PROGRAM INDEXING
VAR
	bStartInput : BOOL;
	bServoOn : BOOL;
	bProgram0_On : BOOL;
	bProgram1_On : BOOL :=TRUE;
	bProgram2_On : BOOL :=FALSE;
	bProgram3_On : BOOL:=FALSE;
	bProgram4_On : BOOL:=FALSE;	
	bHomePositionReturn : BOOL;
	bResetInput : BOOL;
	bEmergencyInput : BOOL := TRUE;
	
	IN_POSITION_INPUT: BOOL;
	IN_POSITIONING_COMPLETION: BOOL;
	IN_START_INPUT_WAIT: BOOL;
	IN_ALARM1: BOOL;
	IN_ALARM2: BOOL;
	IN_READY_STATE: BOOL;
	T1: TON;
	TMR1: TON;
	TMR2: TON;
	TMR3: TON;
	TMR4: TON;
	TMR5: TON;
	TMR6: TON;
	TMR7: TON;
	IN_SERVO_STATUS: BOOL;
	bFirstDigit: BOOL;
	CNT1: CTU;
	ResetCount: BOOL;
	IPC: TP;
	IN_POSITIONING_COMPLET: BOOL;
	CNT2: CTU;
	START_STRAIGTHEN: BOOL;

	START_STRAIGHTEN: R_TRIG;
	START_ROTATING: R_TRIG;
	START_ROTATION: TP;
	SS: R_TRIG;
	CNT_START: CTU;
	TMR_PROCESS: TOF;
	TMR8: TON;
	TMR_OFF: TON;
	TMR_RELEASE: TON;
	INPOS: R_TRIG;
	A: BOOL;
END_VAR

INDEXING_1_VAR.DataByteOutput[0].0 := bProgram0_On;
INDEXING_1_VAR.DataByteOutput[0].1 := bProgram1_On;
INDEXING_1_VAR.DataByteOutput[0].2 := bProgram2_On;
INDEXING_1_VAR.DataByteOutput[0].3 := bProgram3_On;
INDEXING_1_VAR.DataByteOutput[0].4 := bProgram4_On;
INDEXING_1_VAR.DataByteOutput[0].6 := bResetInput;
INDEXING_1_VAR.DataByteOutput[0].7 := bHomePositionReturn;
INDEXING_1_VAR.DataByteOutput[1].0 := bStartInput;
INDEXING_1_VAR.DataByteOutput[1].1 := bServoOn;
INDEXING_1_VAR.DataByteOutput[1].2 := bFirstDigit;
INDEXING_1_VAR.DataByteOutput[1].4 := bEmergencyInput;

IN_POSITION_INPUT := 			INDEXING_1_VAR.DataByteInput [1].0;
IN_POSITIONING_COMPLETION := 	INDEXING_1_VAR.DataByteInput [1].1;
IN_START_INPUT_WAIT := 			INDEXING_1_VAR.DataByteInput [1].2;
IN_ALARM1 := 					INDEXING_1_VAR.DataByteInput [1].3;
IN_ALARM2 := 					INDEXING_1_VAR.DataByteInput [1].4;
IN_READY_STATE :=				INDEXING_1_VAR.DataByteInput [1].7;
IN_SERVO_STATUS :=				INDEXING_1_VAR.DataByteInput [1].6; 
(*
//SERVO ON
IF NOT IN_SERVO_STATUS THEN
	bResetInput := TRUE;
	TMR4(IN:=bResetInput,PT:=T#0.5S);
	IF TMR4.Q THEN
		bResetInput := FALSE;
	END_IF
	bServoOn:=TRUE;
	//POWER_CONTROL.O_PWR_CTRL_INDEXING_1:=TRUE;
	TMR8(IN:=POWER_CONTROL.O_PWR_CTRL_INDEXING_1,PT:=T#0.5S);	
	IF TMR8.Q THEN
		POWER_CONTROL.O_PWR_CTRL_INDEXING_1:=FALSE;
		TMR8(IN:=FALSE);
	END_IF
END_IF
*)
//ALARM RESET
IF NOT IN_ALARM1 OR NOT IN_ALARM2 THEN
	bResetInput := TRUE;
	TMR4(IN:=bResetInput,PT:=T#0.5S);
	INPUT_VAR.ALARM1:=NOT IN_ALARM1 OR NOT IN_ALARM2;
	IF TMR4.Q THEN
		bResetInput := FALSE;
	END_IF
ELSE
	TMR4(IN:=FALSE);
END_IF

IF INDEXING_1_VAR.I_INDEXING_1_ROTATION_DONE THEN
		INDEXING_1_VAR.I_INDEXING_1_HOME:=TRUE;
		bHomePositionReturn:=FALSE;
		//INDEXING_1_VAR.I_INDEXING_1_ROTATION_DONE:=TRUE;
END_IF
//homing
IF NOT INDEXING_1_VAR.I_INDEXING_1_HOME THEN
	bHomePositionReturn:=TRUE;
 	ResetCount:=TRUE;
	INDEXING_1_VAR.O_ROTATION_START:=FALSE;
	INDEXING_1_VAR.I_INDEXING_1_ROTATION_DONE:=FALSE;
	
	INPUT_G6_VAR.O_G6_GRIPPER_EXT_DOWN_1:=FALSE;
	INPUT_G6_VAR.O_G6_GRIPPER_EXT_UP_1:=TRUE;
	
	INPUT_G6_VAR.O_G6_GRIPPER_EXT_DOWN_2:=FALSE;
	INPUT_G6_VAR.O_G6_GRIPPER_EXT_UP_2:=TRUE;
	
	INPUT_G6_VAR.O_G6_GRIPPER_EXT_DOWN_3:=FALSE;
	INPUT_G6_VAR.O_G6_GRIPPER_EXT_UP_3:=TRUE;
	
	INPUT_G6_VAR.O_G6_GRIPPER_EXT_DOWN_4:=FALSE;
	INPUT_G6_VAR.O_G6_GRIPPER_EXT_UP_4:=TRUE;
END_IF



IF (bHomePositionReturn OR bprogram0_on) AND NOT INDEXING_1_VAR.I_INDEXING_1_ROTATION_DONE THEN
	TMR_OFF(IN:=TRUE,PT:=T#40S);
	IF TMR_OFF.Q THEN
		POWER_CONTROL.O_PWR_CTRL_INDEXING_1:=TRUE;
		TMR_RELEASE(IN:=TRUE,PT:=T#0.5S);
		bHomePositionReturn:=FALSE;
	
	END_IF
ELSE
	TMR_OFF(IN:=FALSE);
	TMR_RELEASE(IN:=FALSE);
END_IF
IF TMR_RELEASE.Q THEN
	POWER_CONTROL.O_PWR_CTRL_INDEXING_1:=FALSE;
	TMR_OFF(IN:=FALSE);
END_IF
//start indexing
START_ROTATING(CLK:=INDEXING_1_VAR.O_ROTATION_START);
IF INDEXING_1_VAR.O_ROTATION_START AND IN_START_INPUT_WAIT AND INDEXING_1_VAR.I_INDEXING_1_HOME AND INPUT_VAR.STRAIGHTEN_DONE  THEN
	INDEXING_1_VAR.READY_STRAIGTHEN:=TRUE;
	ELSE
	INDEXING_1_VAR.READY_STRAIGTHEN:=FALSE;	
END_IF

START_ROTATION(IN:=INDEXING_1_VAR.READY_STRAIGTHEN,PT:=T#0.5S);
IF 	START_ROTATION.Q AND NOT TMR_PROCESS.Q AND INDEXING_1_VAR.I_PRESS_STOPPER_UP AND NOT INPUT_G6_VAR.I_G6_START_PLACING AND NOT LOADER_RS4_VAR.I_LOADER_RS4_START_TAKEUP AND INPUT_VAR.STRAIGHTEN_DONE AND NOT INPUT_G6_VAR.I_G6_START_PLACING AND NOT LOADER_RS4_VAR.I_LOADER_RS4_START_TAKEUP THEN
	bprogram0_on:=TRUE;
	IF bprogram0_on THEN
		INDEXING_1_VAR.O_ROTATION_START:=FALSE;
	END_IF
	INDEXING_1_VAR.I_INDEXING_1_ROTATION_DONE:=FALSE;
	IN_POSITIONING_COMPLET :=FALSE;
END_IF
IF bprogram0_on THEN
		A:=FALSE;
	TMR_PROCESS(IN:=TRUE,PT:=T#3S);
	INDEXING_1_VAR.O_ROTATION_START:=FALSE;
	INDEXING_1_VAR.I_INDEXING_1_ROTATION_DONE:=FALSE;
ELSE
	TMR_PROCESS(IN:=FALSE);
END_IF
//select Program No.
IF bprogram0_on AND INDEXING_1_VAR.I_PRESS_STOPPER_UP AND NOT INPUT_G6_VAR.I_G6_START_PLACING AND NOT LOADER_RS4_VAR.I_LOADER_RS4_START_TAKEUP  THEN
	TMR1(IN:=bprogram0_on,PT:=T#15MS);
	bStartInput:=tmr1.Q ;
	IF tmr1.Q THEN
		TMR2(in:=TRUE,pt:=T#25MS);
	END_IF
	IF tmr2.Q THEN
		tmr1(in:=FALSE);
		bStartInput:=FALSE;
	END_IF
	tmr3(in:=tmr2.Q,pt:=T#5MS);
	IF tmr3.Q THEN
		bprogram0_on:= FALSE;
		tmr2(in:=FALSE);
		tmr3(in:=FALSE);
	END_IF
END_IF

IPC(IN:=IN_POSITIONING_COMPLETION,PT:=T#0.01S);
INPOS(CLK:=IN_POSITIONING_COMPLETION);
IF INPOS.Q OR  IN_POSITIONING_COMPLETION THEN
	A:=TRUE;
	IN_POSITIONING_COMPLET :=TRUE;
	INDEXING_1_VAR.I_INDEXING_1_ROTATION_DONE:=TRUE;
END_IF
IF A THEN
	IN_POSITIONING_COMPLET :=TRUE;
	INDEXING_1_VAR.I_INDEXING_1_ROTATION_DONE:=TRUE;
END_IF
IF 	IN_POSITIONING_COMPLET THEN
	INDEXING_1_VAR.I_INDEXING_1_ROTATION_DONE:=TRUE;
END_IF
//IF INDEXING_1_VAR.I_PRESS_STOPPER_UP AND INDEXING_1_VAR.I_INDEXING_1_ROTATION_DONE THEN
IF INDEXING_1_VAR.I_INDEXING_1_ROTATION_DONE THEN
	SS(CLK:=INDEXING_1_VAR.I_INDEXING_1_ROTATION_DONE );
	CNT_START(CU:=SS.Q,RESET:= CNT_START.Q,PV:=2);
	IN_POSITIONING_COMPLET :=FALSE;
	//IF CNT_START.CV=1 THEN
		INPUT_VAR.STRAIGHTEN_START:=SS.Q;
	//END_IF
ELSE
	SS(CLK:=FALSE);
END_IF

IF INPUT_G6_VAR.I_G6_START_PLACING OR LOADER_RS4_VAR.I_LOADER_RS4_START_TAKEUP THEN
	bprogram0_on:= FALSE;
	bStartInput:=FALSE;
END_IF

END_PROGRAM

(* stored: Version 1.1.0.1, ProductVersion 3.1.4020.12
   POU INDEXING: Id {c52200bb-0bf3-4685-b1cf-08b592abb097}, SpecialFunc None *)
